// TIA Portal project "Parcel-locker-siemensS7" (V16)

(* hardware
DEVICE "S71500/ET200MP station_1"  S7-1500 station
   slot 0: "Rail_0"  Rack  6ES7 590-1***0-0AA0
   slot 1: "PLC_1"  CPU 1512C-1 PN  6ES7 512-1CK01-0AB0  V2.8
      slot 3: "CPU display_1"  6ES7591-1AA00-0AA0
      slot 32768: "PROFINET interface_1"  X1
         slot 32769: "Port_1"  X1 P1
         slot 32770: "Port_2"  X1 P2
      slot 34817: "Virtual CP interface port_1"  Virtual CP interface port  Virtual CP interface port
*)

// ===== PLC "PLC_1"  CPU 1512C-1 PN =====

VAR_GLOBAL   // PLC tag table "Default tag table"
   "Box1" AT %Q0.0 : Bool;
   "Box2" AT %Q0.1 : Bool;
   "Box3" AT %Q0.2 : Bool;
END_VAR

// folder: Common

TYPE "typeDiagnostics"
TITLE = typeDiagnostics
// Provides a structure for detailed diagnostics
   STRUCT
      status : Word;   // Status of the block or error identification when error occurred
      subfunctionStatus : DWord;   // Status or return value of called FBs, FCs and system blocks
      stateNumber : DInt;   // State in the state machine of the block where the error occurred
   END_STRUCT;
END_TYPE

// folder: LHTTP

TYPE "LHTTP_typeTLS"
   STRUCT
      validateServerIdentity : Bool;   // Validate the subjectAlternateName in the X.509-V3 certificate of the server to check the identity of the server
      serverCert : UDInt;   // ID of the X.509-V3 certificate (usually a CA certificate) that is used by the TLS client to validate the TLS server authentication. If this parameter is 0, the TLS client uses all (CA) certificates currently loaded in the client certificate store to validate the server authentication.
      clientCert : UDInt;   // ID of own X.509 V3 certificate
   END_STRUCT;
END_TYPE

// folder: (top level)

DATA_BLOCK "Modbus_server_parameters"   // DB2
{ S7_Optimized_Access := 'TRUE' }
VERSION : 0.1
   VAR
      NDR : Bool;
      DR : Bool;
      ERROR : Bool;
      STATUS : Word;
      CONNECT : TCON_IP_v4;
   END_VAR
BEGIN
   CONNECT.InterfaceId := 64;
   CONNECT.ID := 1;
   CONNECT.LocalPort := 502;
END_DATA_BLOCK

DATA_BLOCK "Modbus_data"   // DB3
{ S7_Optimized_Access := 'FALSE' }
VERSION : 0.1
   VAR
      Boxes : Array[0..3] of Int;
   END_VAR
BEGIN
END_DATA_BLOCK

DATA_BLOCK "Modbus_server_DB"   // DB4
{ S7_Optimized_Access := 'TRUE' }
VERSION : 0.1
// stored: InstanceOfName Modbus_server
"Modbus_server"
BEGIN
END_DATA_BLOCK

FUNCTION_BLOCK "Modbus_server"   // FB1, LAD
{ S7_Optimized_Access := 'TRUE' }
VERSION : 0.1
BEGIN

REGION Network 1
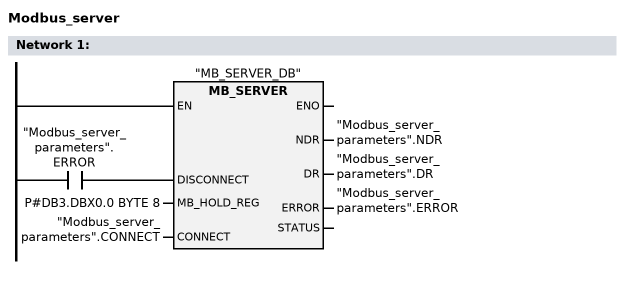
   "MB_SERVER_DB"(DISCONNECT := "Modbus_server_parameters".ERROR,   // MB_SERVER
                  MB_HOLD_REG := P#DB3.DBX0.0 BYTE 8,
                  CONNECT := "Modbus_server_parameters".CONNECT,
                  NDR => "Modbus_server_parameters".NDR,
                  DR => "Modbus_server_parameters".DR,
                  ERROR => "Modbus_server_parameters".ERROR);
END_REGION
END_FUNCTION_BLOCK

ORGANIZATION_BLOCK "Main"   // OB1, LAD, ProgramCycle
TITLE = "Main Program Sweep (Cycle)"
{ S7_Optimized_Access := 'TRUE' }
VERSION : 0.1
   VAR_INPUT
      Initial_Call : Bool;   // Initial call of this OB
      Remanence : Bool;   // =True, if remanent data are available
   END_VAR
BEGIN

REGION Network 1
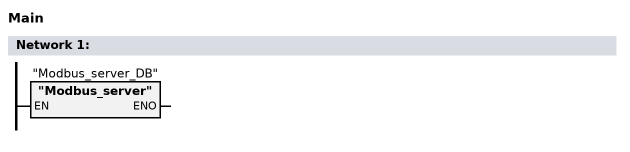
   RUNG wire#powerrail
      "Modbus_server_DB"()
   END_RUNG
   // the same network as SCL:
   "Modbus_server_DB"();   // "Modbus_server"
END_REGION

REGION Network 3 (SCL)
   // Open Box1
   IF ("Modbus_data".Boxes[0] AND 2#0000_0000_0000_0001) <> 0 THEN
       "Box1" := TRUE;
   ELSE
       "Box1" := FALSE;
   END_IF;
END_REGION

REGION Network 4 (SCL)
   // Open Box2
   IF ("Modbus_data".Boxes[0] AND 2#0000_0000_0000_0010) <> 0 THEN
       "Box2" := TRUE;
   ELSE
       "Box2" := FALSE;
   END_IF;
END_REGION

REGION Network 5 (SCL)
   // Open Box3
   IF ("Modbus_data".Boxes[0] AND 2#0000_0000_0000_0100) <> 0 THEN
       "Box3" := TRUE;
   ELSE
       "Box3" := FALSE;
   END_IF;
END_REGION
END_ORGANIZATION_BLOCK

// ===== library types =====

// folder: LHTTP

FUNCTION_BLOCK "LHTTP_Get"   // FB8, SCL
TITLE = LHTTP_Get
{ S7_Optimized_Access := 'TRUE' }
AUTHOR : SIOS
FAMILY : LHTTP
VERSION : 2.1
// Implements the HTTP GET method
   VAR_INPUT
      execute : Bool;   // Send HTTP request
      hwID : Hw_Any;   // Hardware ID of Ethernet interface
      connID : Conn_Ouc := 1;   // Unique connection ID
      url : String;   // URL, i.e. "http://www.siemens.com/simatic"
      queryParams : String;   // Additional query parameters if "url" is not long enough, i.e. "lang=en&q=simatic"; "?" or "&" is inserted automatically in between "url" and "queryParameters". / Optional query parameters that are appended to URL, i.e. "lang=en&q=simatic"
      userFields : Array[0..#UPPER_USER_FIELDS] of Char;   // Additional user-defined header fields
      tls : "LHTTP_typeTLS";   // TLS certificates for secure connections (HTTPS), leave open for non-secure connections (HTTP)
      keepConnection : Bool;   // Keep connection established after execution of request
      timeOut : Time := T#10s;   // Time to wait for response from server
   END_VAR
   VAR_OUTPUT
      connected : Bool;   // Connection to web server is established
      done : Bool;   // HTTP request finished
      busy : Bool;   // Function is busy
      error : Bool;   // An error occured
      status : Word := 16#7000;   // Specifies the error
      diagnostics : "typeDiagnostics";   // Diagnostics information of FB
      responseCode : UInt;   // HTTP response code
      length : UDInt;   // Length of received data
   END_VAR
   VAR_IN_OUT
      responseData : Array[*] of Char;   // Data received from HTTP server
   END_VAR
   VAR
      instTSendC : TSEND_C;   // Instance of TSEND_C
      instTRcv : TRCV;   // Instance of TRCV
      instTimeout : TON_TIME;   // Time-out
      statConnected : Bool;   // Static value for output 'connected'
      statDone : Bool;   // Static value for output 'done'
      statBusy : Bool;   // Static value for output 'busy'
      statError : Bool;   // Static value for output 'error'
      statStatus : Word := 16#7000;   // Static value for output 'status'
      statResponseCode : UInt;   // Static value for output 'responseCode'
      statLength : UDInt;   // Static value for output 'length'
      statFBState : USInt := 0;   // Current state in state machine
      statSubfunctionStatus : DWord;   // Status or return value of called FBs, FCs and system blocks
      statEmptyDiagnostics : "typeDiagnostics";   // Empty diagnostics information (for initialization purposes only)
      statParam : Struct   // Connection parameters
         isQDN : Bool;
         paramQDN : TCON_QDN_SEC;   // Connection parameters in form of QDN
         paramIP : TCON_IP_V4_SEC;   // Connection parameters in form of IP address
      END_STRUCT;
      statHost : String;   // Host part of URL
      statRequest : Struct   // GET request
         chars : Array[0..#UPPER_REQUEST_ARRAY] of Char;   // GET request (max. length: url (254) + data (254) + header (94)
         length : UInt;   // Length of GET request
      END_STRUCT;
      statSend : Struct   // Parameters for instruction TSend_C
         connect : Bool;   // Establish and keep connection
         req : Bool;   // Send data
      END_STRUCT;
      statEncoding : String;   // Transfer encoding of response from HTTP server
      statContentLength : UInt;   // Content length as specified in header of response
      statChunkLen : UDInt;   // Remaining length of current chunk
      statRcvdLen : UDInt;   // Sum length of received data
      statTimeoutIn : Bool;   // Timeout
      statRcvBuffer : Array[0..#UPPER_TCP_FRAME] of Char;   // Temporary receive buffer
      statSizeRcvArray : UDInt;   // Size of receive buffer at parameter "responseData"
      statExecuteOld : Bool;   // Last cycle's value of input "execute"
   END_VAR
   VAR_TEMP
      tempUrl : String;   // Copy of URL
      tempQuery : String;   // Query part of URL
      tempIndex : DInt;   // Index for for loops
      tempPos : Int;   // General tag for positions
      tempLen : UInt;   // General tag for lengths
      tempRet : Word;   // General tag for return values
      tempString : String;   // General tag for strings
      tempExitLoop : Bool;   // Condition to exit REPEAT loop around state machine
      tempChunk : Struct   // Temporary tags for chunked encoding
         posData : UInt;   // Start position of data in current packet
         lenData : UInt;   // Length of data in current packet
         exitLoop : Bool;   // Condition to exit loop
      END_STRUCT;
   END_VAR
   VAR CONSTANT
      UPPER_REQUEST_ARRAY : UInt := 1459;   // Upper limit of request array
      UPPER_TCP_FRAME : UInt := 1459;   // Upper limit of a TCP/IP frame
      UPPER_USER_FIELDS : USInt := 255;   // Upper limit of userFields
      PORT_UNSECURE : UInt := 80;   // Port for unsecure HTTP connection
      PORT_SECURE : UInt := 443;   // Port for secure HTTP connection
      POS_RESPONSE_CODE : USInt := 9;   // Position of HTTP response code in response message
      STATUS_DONE : Word := 16#0000;   // Job finished without errors
      STATUS_DISCONNECTED : Word := 16#0003;   // Communication connection closed
      STATUS_IDLE : Word := 16#7000;   // No job
      STATUS_FIRST_CALL : Word := 16#7001;   // First call after incoming new job (rising edge 'execute')
      STATUS_CONNECTING : Word := 16#7002;   // Connection is currently being established
      STATUS_DISCONNECTING : Word := 16#7003;   // Communication connection is being terminated
      STATUS_MONITORING : Word := 16#7004;   // Communication connection has been established and is being monitored. No send job execution active
      STATUS_SENT : Word := 16#7005;   // Request sent, waiting for response
      SUB_STATUS_NO_ERROR : DWord := 16#0000_0000;   // No error occured in subfunction call
      ERR_BOUND_NOT_ZERO : Word := 16#8201;   // Lower bound of receive buffer is not 0
      ERR_INVALID_URL : Word := 16#8202;   // Invalid URL
      ERR_DIFFERENT_HOST : Word := 16#8203;   // Trying to use existing connection with different host
      ERR_END_USER_FIELDS : Word := 16#8206;   // End of user-defined header fields could not be found
      ERR_REQUEST_SIZE : Word := 16#8210;   // Request array is too small for specified parameters
      ERR_RESPONSE_SIZE : Word := 16#8220;   // Receive buffer at parameter "responseData" too small
      ERR_CONN_LOST : Word := 16#8400;   // Offset for lost connection
      ERR_FORWARDING : Word := 16#8403;   // Server responded with forwarding message. Forwarding is not supported, see "diagnostics"
      ERR_WEBSERVER : Word := 16#8404;   // Webserver responded with error code, see "diagnostics"
      ERR_INVALID_HEADER : Word := 16#8405;   // Header of response is invalid
      ERR_TIMEOUT : Word := 16#8408;   // Time-out occurred
      ERR_UNDEFINED_STATE : Word := 16#8600;   // Error due to an undefined state in state machine
      ERR_TSENDC : Word := 16#8601;   // Error: TCON encountered an error, see "diagnostics"
      ERR_TRCV : Word := 16#8603;   // Error: TURCV encountered error, see "diagnostics"
      ERR_MOVE_USER_FIELDS : Word := 16#8612;   // Error in MOVE_BLK_VARIANT to copy user-defined header fields, see "diagnostics"
      ERR_ENCODING_UNKNOWN : Word := 16#8620;   // Transfer encoding of response could not be detected or is unsupported
      ERR_MOVE_IDENTITY : Word := 16#8630;   // Error in MOVE_BLK_VARIANT for transfer encoding 'identity', see "diagnostics"
      ERR_DECODING_FAILED : Word := 16#8640;   // Chunk encoded response could not be decoded
      ERR_MOVE_CHUNKED : Word := 16#8641;   // Error in MOVE_BLK_VARIANT for transfer encoding 'chunked', see "diagnostics"
      TSENDC_STATUS_CONNECTED : Word := 16#0001;   // TSEND_C: Communication connection established
      MOVE_STATUS_SIZE : Word := 16#8483;   // MOVE_BLK_VARIANT: DEST too small
      FB_STATE_NO_PROCESSING : USInt := 0;   // FB state: No processing
      FB_STATE_INIT : USInt := 1;   // FB state: initialization
      FB_STATE_REQUEST : USInt := 2;   // FB state: prepare request
      FB_STATE_SEND : USInt := 3;   // FB state: send request
      FB_STATE_RCV : USInt := 4;   // FB state: receive data
      FB_STATE_MON : USInt := 5;   // FB state: monitoring connection
      CRLF : String := '$R$L';   // Newline control character (carriage return, line feed)
      HEADER_END : String := '$R$L$R$L';   // End of HTTP header (two newline control characters)
      LEN_CRLF : UInt := 2;   // Length of CRLF
   END_VAR
   // statParam.paramIP.ConnPara.ActiveEstablished := true;
   // statParam.paramQDN.ConnPara.ActiveEstablished := true;
BEGIN
   REGION BLOCK INFO HEADER
     //===============================================================================
     // SIEMENS / (c)Copyright 2021
     //-------------------------------------------------------------------------------
     // Title:        LHTTP_Get
     // Function:     Implements the HTTP GET method
     // Library:      LHTTP
     // Author:       Siemens Industry Online Support
     // Tested with:  CPU 1516-3 PN/DP V2.8
     // Engineering:  TIA Portal V16
     // Restrictions: --
     // Requirements: S7-1200 with firmware V4.4 or higher
     //               S7-1500 with firmware V2.0 or higher
     //-------------------------------------------------------------------------------
     // Change log table:
     // Version  | Date       | Expert in charge       | Changes applied
     //----------|------------|------------------------|------------------------------
     // 02.01.00 | 2021-12-15 | Online Support         | Renamed parameter "data" to "queryParams"
     //-------------------------------------------------------------------------------
     // 02.00.04 | 2021-05-10 | Online Support         | Fixed issues with chunked encoding
     //          |            |                        | Allow chunk sizes > 65535 Bytes
     //          |            |                        | Made header evaluation case-insensitive
     //-------------------------------------------------------------------------------
     // 02.00.00 | 2020-12-16 | Online Support         | Added option to keep connection established
     //          |            |                        | Added parameter to add user-defined headers fields
     //          |            |                        | Changed to data type of "data" to Variant to allow larger data
     //          |            |                        | Removed "statusID" and added "diagnostics" instead, changed some error codes
     //-------------------------------------------------------------------------------
     // 01.00.00 | 2019-04-01 | Online Support         | First released version
     //===============================================================================
   END_REGION

   REGION INSTRUCTIONS
     IF (#statStatus <> #STATUS_IDLE) THEN // Only execute when FB is triggered to reduce system load
       // Connect and send
       IF #statParam.isQDN THEN // Call if host is a domain name
         #instTSendC(REQ     := #statSend.req,
                     CONT    := #statSend.connect,
                     LEN     := #statRequest.length,
                     CONNECT := #statParam.paramQDN,
                     DATA    := #statRequest.chars);
       ELSE // Call if host is an IP address
         #instTSendC(REQ     := #statSend.req,
                     CONT    := #statSend.connect,
                     LEN     := #statRequest.length,
                     CONNECT := #statParam.paramIP,
                     DATA    := #statRequest.chars);
       END_IF;

       // Receive
       #instTRcv(ID    := #statParam.paramQDN.ConnPara.ID,
                 EN_R  := #statFBState >= #FB_STATE_RCV,
                 LEN   := 0,
                 ADHOC := true,
                 DATA  := #statRcvBuffer);

       // Monitor time out
       #instTimeout(IN := #statTimeoutIn,
                    PT := #timeOut);

       IF #instTimeout.Q THEN
         #statStatus := #ERR_TIMEOUT;
       END_IF;
     END_IF;
   END_REGION

   REGION TRIGGERING
     IF (#execute = true AND #statExecuteOld = false) // Check if FB is triggered
       AND (#statStatus = #STATUS_IDLE OR #statStatus = #STATUS_MONITORING)
     THEN // First call; initialize FB
       // Copy URL
       #tempUrl := #url;

       #statBusy := true;
       #statStatus := #STATUS_FIRST_CALL;
       #statSubfunctionStatus := #SUB_STATUS_NO_ERROR;
       #diagnostics := #statEmptyDiagnostics;

       IF #statConnected = FALSE THEN // Connection is not yet established
         #statFBState := #FB_STATE_INIT;
       ELSE // Connection is already established, skip init
         #statFBState := #FB_STATE_REQUEST;
       END_IF;

     ELSIF (#statStatus = #STATUS_FIRST_CALL) THEN
       #statStatus := #STATUS_CONNECTING;
     END_IF;

     // Edge detection 'execute' input
     #statExecuteOld := #execute;
   END_REGION TRIGGERING

   IF (#statStatus = #STATUS_IDLE) THEN // Nothing to do -> End here to reduce "system load"
     RETURN;
   END_IF;

   REGION STATE_MACHINE
     // State machine is wrapped in REPEAT loop to make it possible to quickly exit state machine
     // in case of an error or to go through CASE multiple times within one cycle
     REPEAT
       #tempExitLoop := true; // Condition to exit loop is set per default

       CASE #statFBState OF // State machine of FB
         #FB_STATE_NO_PROCESSING: // No processing active
           ;

         #FB_STATE_INIT:
           REGION INIT
             // Get size of receive buffer
             IF LOWER_BOUND(ARR := #responseData, DIM := 1) <> 0 THEN
               #statStatus := #ERR_BOUND_NOT_ZERO;
               EXIT;
             ELSE
               #statSizeRcvArray := DINT_TO_UDINT(UPPER_BOUND(ARR := #responseData, DIM := 1)) + 1;
             END_IF;

             // Set connection parameters
             #statParam.paramQDN.ConnPara.InterfaceId := #hwID;
             #statParam.paramQDN.ConnPara.ID := #connID;
             #statParam.paramIP.ConnPara.InterfaceId := #hwID;
             #statParam.paramIP.ConnPara.ID := #connID;

             // Check if network protocol was specified to determine if connection should be secured
             #tempPos := FIND(IN1 := #tempUrl, IN2 := 'https://');
             IF #tempPos = 1 THEN // HTTPS
               #statParam.paramQDN.ActivateSecureConn := true;
               #statParam.paramQDN.ExtTLSCapabilities.%X0 := #tls.validateServerIdentity;
               #statParam.paramQDN.TLSServerCertRef := #tls.serverCert;
               #statParam.paramQDN.TLSClientCertRef := #tls.clientCert;
               #statParam.paramIP.ActivateSecureConn := true;
               #statParam.paramIP.ExtTLSCapabilities.%X0 := #tls.validateServerIdentity;
               #statParam.paramIP.TLSServerCertRef := #tls.serverCert;
               #statParam.paramIP.TLSClientCertRef := #tls.clientCert;
               // Delete network protocol from URL
               #tempUrl := DELETE(IN := #tempUrl, L := 8, P := 1);
             ELSE // HTTP
               #statParam.paramQDN.ActivateSecureConn := false;
               #statParam.paramIP.ActivateSecureConn := false;
               // Delete network protocol from URL if specified
               IF #tempUrl[5] = ':' THEN
                 #tempUrl := DELETE(IN := #tempUrl, L := 7, P := 1);
               END_IF;
             END_IF;

             // Determine if host is domain name or IP address
             #tempPos := CHAR_TO_INT(#tempUrl[1]);
             IF #tempPos >= CHAR_TO_INT('A') AND #tempPos <= CHAR_TO_INT('z') THEN // Host is a domain name
               #statParam.isQDN := true;
             ELSIF #tempPos >= CHAR_TO_INT('0') AND #tempPos <= CHAR_TO_INT('9') THEN // Host is an IP address
               #statParam.isQDN := false;
             ELSE // URL invalid
               #statStatus := #ERR_INVALID_URL;
               EXIT;
             END_IF;

             // Get host name and port
             #tempPos := FIND(IN1 := #tempUrl, IN2 := '/');
             IF #tempPos > 0 THEN // URL has a path after host name
               #statHost := LEFT(IN := #tempUrl, L := #tempPos - 1);
             ELSE
               #statHost := #tempUrl;
             END_IF;
             #tempPos := FIND(IN1 := #statHost, IN2 := ':');
             IF #tempPos > 0 THEN // Port specified in URL
               #statParam.paramQDN.ConnPara.RemotePort := STRING_TO_UINT(DELETE(IN := #statHost, L := #tempPos, P := 1));
               #statParam.paramIP.ConnPara.RemotePort := STRING_TO_UINT(DELETE(IN := #statHost, L := #tempPos, P := 1));
               #statHost := LEFT(IN := #statHost, L := #tempPos - 1);
             ELSE // No port specified in URL, set default port
               IF #statParam.paramQDN.ActivateSecureConn OR #statParam.paramIP.ActivateSecureConn THEN
                 #statParam.paramQDN.ConnPara.RemotePort := #PORT_SECURE;
                 #statParam.paramIP.ConnPara.RemotePort := #PORT_SECURE;
               ELSE
                 #statParam.paramQDN.ConnPara.RemotePort := #PORT_UNSECURE;
                 #statParam.paramIP.ConnPara.RemotePort := #PORT_UNSECURE;
               END_IF;
             END_IF;

             IF #statParam.isQDN THEN // Host is a domain name
               #statParam.paramQDN.ConnPara.RemoteQDN := CONCAT(IN1 := #statHost, IN2 := '.');
             ELSE // Host is an IP address
               #tempString := #statHost;
               FOR #tempIndex := 1 TO 3 DO
                 #tempPos := FIND(IN1 := #tempString, IN2 := '.');
                 #statParam.paramIP.ConnPara.RemoteAddress.ADDR[#tempIndex] := UINT_TO_BYTE(STRING_TO_UINT(LEFT(IN := #tempString, L := #tempPos - 1)));
                 #tempString := DELETE(IN := #tempString, L := #tempPos, P := 1);
               END_FOR;
               #statParam.paramIP.ConnPara.RemoteAddress.ADDR[4] := UINT_TO_BYTE(STRING_TO_UINT(#tempString));
             END_IF;

             #statFBState := #FB_STATE_REQUEST;
             #tempExitLoop := FALSE; // Don't exit loop to go directly to prepare request
           END_REGION INIT

         #FB_STATE_REQUEST:
           REGION PREP_REQUEST
             // Check host in URL when using existing connection
             IF #statConnected = TRUE THEN
               #tempPos := FIND(IN1 := #tempUrl, IN2 := #statHost);
               IF #tempPos = 0 THEN // URL doesn't contain expected host
                 #statStatus := #ERR_DIFFERENT_HOST;
                 EXIT;
               ELSE // Scheme and host must be deleted for further processing
                 #tempUrl := DELETE(IN := #tempUrl, L := #tempPos + LEN(#statHost) - 1, P := 1);
               END_IF;
             END_IF;

             // Get path
             #tempPos := FIND(IN1 := #tempUrl, IN2 := '/');
             IF #tempPos > 0 THEN // URL has a path after host name
               #tempString := DELETE(IN := #tempUrl, L := #tempPos - 1, P := 1);
             ELSE
               #tempString := '/';
             END_IF;

             // Prepare query part of URL
             IF #queryParams <> '' THEN // Parameter is in use
               IF #queryParams[1] = '?' OR #queryParams[1] = '&' THEN
                 #tempQuery := DELETE(IN := #queryParams, P := 1, L := 1);
               ELSE
                 #tempQuery := #queryParams;
               END_IF;
               #tempPos := FIND(IN1 := #tempString, IN2 := '?'); // Check if URL already contains query parameters
               IF #tempPos <> 0 THEN // URL already contains query parameters
                 #tempQuery := CONCAT(IN1 := '&', IN2 := #tempQuery); // Append query parameters with &
               ELSE // URL does not contain query parameters
                 #tempQuery := CONCAT(IN1 := '?', IN2 := #tempQuery); // Append query parameters with ?
               END_IF;
             END_IF;

             // Put together GET request
             // Strg_TO_Chars conversion is done several times to utilize maximum length of parameters url and query parameters
             Strg_TO_Chars(Strg   := CONCAT(IN1 := 'GET ', IN2 := #tempString), // Path cannot be longer than 249 characters --> save to use CONCAT
                           pChars := 0,
                           Cnt    => #tempLen,
                           Chars  := #statRequest.chars);
             #tempPos := UINT_TO_INT(#tempLen);

             Strg_TO_Chars(Strg   := #tempQuery,
                           pChars := #tempPos,
                           Cnt    => #tempLen,
                           Chars  := #statRequest.chars);
             #tempPos += UINT_TO_INT(#tempLen);

             Strg_TO_Chars(Strg   := CONCAT(IN1 := ' HTTP/1.1$R$LHost: ', IN2 := #statHost), // Host will not use all 254 characters --> save to use CONCAT
                           pChars := #tempPos,
                           Cnt    => #tempLen,
                           Chars  := #statRequest.chars);
             #tempPos += UINT_TO_INT(#tempLen);

             Strg_TO_Chars(Strg   := '$R$LUser-Agent: SIMATIC Controller (LHTTP)$R$LAccept: text/html$R$LAccept-Encoding: identity$R$LAccept-Charset: utf-8$R$L',
                           pChars := #tempPos,
                           Cnt    => #tempLen,
                           Chars  := #statRequest.chars);
             #tempPos += UINT_TO_INT(#tempLen);

             // Insert additional user-defined header fields
             IF #userFields[0] <> ' ' THEN
               FOR #tempLen := 0 TO #UPPER_USER_FIELDS DO
                 IF #userFields[#tempLen] = '$00' THEN
                   EXIT;
                 END_IF;
               END_FOR;

               IF #tempLen > #UPPER_USER_FIELDS THEN // End not found
                 #statStatus := #ERR_END_USER_FIELDS;
                 EXIT;
               END_IF;

               #tempRet := INT_TO_WORD(MOVE_BLK_VARIANT(SRC := #userFields, COUNT := #tempLen, SRC_INDEX := 0, DEST_INDEX := #tempPos, DEST => #statRequest.chars));

               IF #tempRet = #MOVE_STATUS_SIZE THEN
                 #statStatus := #ERR_REQUEST_SIZE;
                 EXIT;
               ELSIF #tempRet <> 16#0000 THEN
                 #statStatus := #ERR_MOVE_USER_FIELDS;
                 #statSubfunctionStatus := #tempRet;
                 EXIT;
               END_IF;

               #tempPos += UINT_TO_INT(#tempLen);

               // Append CRLF if needed
               IF #statRequest.chars[#tempPos - 2] <> '$R' AND #statRequest.chars[#tempPos - 1] <> '$L' THEN
                 #statRequest.chars[#tempPos] := '$R';
                 #statRequest.chars[#tempPos + 1] := '$L';
                 #tempPos += 2;
               END_IF;
             END_IF;

             // Append end of header section
             Strg_TO_Chars(Strg   := #CRLF,
                           pChars := #tempPos,
                           Cnt    => #tempLen,
                           Chars  := #statRequest.chars);
             #tempPos += UINT_TO_INT(#tempLen);

             // Calculate total length of request
             #statRequest.length := INT_TO_UINT(#tempPos);

             #statSend.connect := true; // Connect
             #statSend.req := true; // Send request
             #statTimeoutIn := true; // Start timer
             #statFBState := #FB_STATE_SEND;
           END_REGION

         #FB_STATE_SEND: // Send data
           REGION SEND
             IF #instTSendC.STATUS = #TSENDC_STATUS_CONNECTED THEN
               #statConnected := TRUE;
             ELSIF #instTSendC.DONE THEN
               #statStatus := #STATUS_SENT;
               #statFBState := #FB_STATE_RCV;
               // Don't exit loop to go directly to receive state
               // without waiting for next cycle so that no responses can be missed
               #tempExitLoop := false;
             ELSIF #instTSendC.ERROR THEN
               #statStatus := #ERR_TSENDC;
               #statSubfunctionStatus := #instTSendC.STATUS;
             END_IF;
           END_REGION

         #FB_STATE_RCV: // Wait for new data
           REGION RCV
             IF #instTRcv.NDR THEN

               REGION HEADER_EVAL
                 // Evaluate header if received packet is first packet
                 IF #statEncoding = '' THEN
                   // Get response code
                   Chars_TO_Strg(Chars  := #statRcvBuffer,
                                 pChars := #POS_RESPONSE_CODE,
                                 Cnt    := 3,
                                 Strg   => #tempString);
                   #statResponseCode := STRING_TO_UINT(#tempString);

                   // Exit loop immediately and output errror if response code shows errors or forwarding
                   IF #statResponseCode >= 300 THEN
                     #tempRet := ATH(IN := #tempString, N := 3, OUT => #statSubfunctionStatus); // Interpret response code as hexadecimal
                     #statSubfunctionStatus := SHR(IN := #statSubfunctionStatus, N := 20);
                     IF #statResponseCode >= 400 THEN
                       #statStatus := #ERR_WEBSERVER;
                     ELSE
                       #statStatus := #ERR_FORWARDING;
                     END_IF;
                     EXIT;
                   END_IF;

                   // Get length of HTTP header
                   #tempLen := DINT_TO_UINT("LHTTP_FindStringInArray"(searchFor := #HEADER_END, searchIn := #statRcvBuffer) + LEN(#HEADER_END));

                   // Exit loop immediately and output errror if header end cannot be found
                   IF #tempLen = 0 THEN
                     #statStatus := #ERR_INVALID_HEADER;
                     EXIT;
                   END_IF;

                   // Search header for content length
                   #tempRet := "LHTTP_ExtractStringFromArray"(textBefore := 'Content-Length: ',
                                                              textAfter := #CRLF,
                                                              extractedString => #tempString,
                                                              searchIn := #statRcvBuffer);

                   IF #tempRet <> 0 THEN // Content length not found; try lower-case
                     #tempRet := "LHTTP_ExtractStringFromArray"(textBefore := 'content-length: ',
                                                                textAfter := #CRLF,
                                                                extractedString => #tempString,
                                                                searchIn := #statRcvBuffer);
                   END_IF;

                   IF #tempRet = 0 THEN // Content length found
                     #statContentLength := STRING_TO_UINT(#tempString);
                     #statEncoding := 'identity';
                   ELSE // Can't detect content length, check if transfer encoding is 'chunked'
                     #tempPos := DINT_TO_INT("LHTTP_FindStringInArray"(searchFor := 'chunked', searchIn := #statRcvBuffer));

                     IF #tempPos >= 0 THEN
                       #statEncoding := 'chunked';
                     ELSE // Exit loop immediately and output error if content length nor transfer encoding can be detected
                       #statStatus := #ERR_ENCODING_UNKNOWN;
                       EXIT;
                     END_IF;
                   END_IF;

                   IF #instTRcv.RCVD_LEN = #tempLen THEN // Packet contains no body, wait for next packet
                     EXIT;
                   END_IF;
                 END_IF;
               END_REGION

               REGION TE_IDENTITY
                 IF #statEncoding = 'identity' THEN // Transfer encoding is 'identity'
                   // Move data from buffer to output; tempLen contains header length during first packet, otherwise 0
                   #tempRet := INT_TO_WORD(MOVE_BLK_VARIANT(SRC := #statRcvBuffer,
                                                                                    COUNT := MIN(IN1 := #instTRcv.RCVD_LEN - #tempLen, IN2 := #statSizeRcvArray - #statRcvdLen), // Move as much as possible to output
                                                                                    SRC_INDEX := #tempLen,
                                                                                    DEST_INDEX := UDINT_TO_DINT(#statRcvdLen),
                                                                                    DEST => #responseData));

                   // Exit loop immediately and output error if data could not be moved
                   IF #tempRet <> 0 THEN
                     #statStatus := #ERR_MOVE_IDENTITY;
                     #statSubfunctionStatus := #tempRet;
                     EXIT;
                   END_IF;

                   // Add length of received packet to sum; tempLen contains header length during first packet, otherwise 0
                   #statRcvdLen += #instTRcv.RCVD_LEN - #tempLen;

                   IF #statRcvdLen > #statSizeRcvArray THEN // Receive buffer too small
                     #statStatus := #ERR_RESPONSE_SIZE;
                     #statLength := #statContentLength; // Output required size of buffer
                   ELSIF #statRcvdLen >= #statContentLength THEN // Everything was received
                     #statStatus := #STATUS_DONE;
                     #statLength := #statRcvdLen;
                   END_IF;
                 END_IF;
               END_REGION

               REGION TE_CHUNKED
                 IF #statEncoding = 'chunked' THEN // Transfer encoding is 'chunked'

                   // Set position of chunk data
                   #tempChunk.posData := #tempLen; // tempLen contains header length during first packet, otherwise 0

                   REPEAT
                     #tempChunk.exitLoop := true; // Condition to exit loop is set per default

                     // Read length of chunk if received packet is first packet or a previous chunk was received completely
                     IF #statChunkLen = 0 THEN
                       // Extract hexadecimal chunk-size field
                       Chars_TO_Strg(Chars  := #statRcvBuffer,
                                     pChars := #tempChunk.posData,
                                     Cnt    := 0,
                                     Strg   => #tempString);
                       #tempPos := FIND(IN1 := #tempString, IN2 := #CRLF);
                       #tempRet := ATH(IN := #tempString, N := #tempPos - 1, OUT => #statChunkLen);
                       // Shift bits to the right depending on length of chunk size, since ATH is left aligned
                       #statChunkLen := SHR(IN := #statChunkLen, N := 4 * INT_TO_UINT(8 - (#tempPos - 1)));

                       // Move start position of data behind chunk-size field
                       #tempChunk.posData += INT_TO_UINT(#tempPos) + 1;

                       // Exit loop immediately and output error if chunk size cannot be detected
                       IF #tempRet <> 0 THEN
                         #statStatus := #ERR_DECODING_FAILED;
                         EXIT;
                       END_IF;
                     END_IF;

                     IF #statChunkLen = 0 THEN // Length was evaluated, chunk contains no data --> final chunk received
                       #statStatus := #STATUS_DONE;
                       #statLength := #statRcvdLen;
                     ELSE // Chunk contains data
                       // Evaluate length of received packet and set length of data accordingly
                       IF #instTRcv.RCVD_LEN = #tempChunk.posData + #statChunkLen + #LEN_CRLF THEN // Chunk was received entirely and packet contains no further chunks
                         #tempChunk.lenData := UDINT_TO_UINT(#statChunkLen); // Output remaining length of chunk
                       ELSIF #instTRcv.RCVD_LEN < #tempChunk.posData + #statChunkLen + #LEN_CRLF THEN // Packet only contains part of chunk
                         #tempChunk.lenData := UDINT_TO_UINT(#instTRcv.RCVD_LEN) - #tempChunk.posData; // Output entire packet without possible chunk-size field
                       ELSIF #instTRcv.RCVD_LEN > #tempChunk.posData + #statChunkLen + #LEN_CRLF THEN // Current packet contains more than one chunk
                         #tempChunk.lenData := UDINT_TO_UINT(#statChunkLen); // Output remaining length of chunk
                         #tempChunk.exitLoop := false; // Execute loop again since packet contains more data
                       ELSE // Can't decode message
                         #statStatus := #ERR_DECODING_FAILED;
                         EXIT;
                       END_IF;

                       // Move received data to output
                       #tempRet := INT_TO_WORD(MOVE_BLK_VARIANT(SRC := #statRcvBuffer,
                                                                                        COUNT := MIN(IN1 := #tempChunk.lenData, IN2 := #statSizeRcvArray - #statRcvdLen), // Move as much as possible to output
                                                                                        SRC_INDEX := #tempChunk.posData,
                                                                                        DEST_INDEX := UDINT_TO_DINT(#statRcvdLen),
                                                                                        DEST => #responseData));

                       // Exit loop immediately and output error if data could not be moved
                       IF #tempRet <> 0 THEN
                         #statStatus := #ERR_MOVE_CHUNKED;
                         #statSubfunctionStatus := #tempRet;
                         EXIT;
                       END_IF;

                       // Move start position of data behind data of current chunk in case packet contains more data; only relevant if REPEAT loop is executed again
                       #tempChunk.posData += #tempChunk.lenData + #LEN_CRLF;

                       // Subtract length of data in current packet from remaining length of chunk and add to sum of received data
                       #statChunkLen -= #tempChunk.lenData;
                       #statRcvdLen += #tempChunk.lenData;

                       IF #statRcvdLen > #statSizeRcvArray THEN // Receive buffer too small
                         #statStatus := #ERR_RESPONSE_SIZE;
                         #statLength := #statRcvdLen; // Output required size of buffer according to so far received chunked messages
                         EXIT;
                       END_IF;
                     END_IF;
                   UNTIL (#tempChunk.exitLoop = true) END_REPEAT;
                 END_IF;
               END_REGION

             ELSIF #instTRcv.ERROR THEN
               #statStatus := #ERR_TRCV;
               #statSubfunctionStatus := #instTRcv.STATUS;
             END_IF;
           END_REGION

         #FB_STATE_MON:
           REGION MONITORING
             IF #keepConnection = FALSE THEN // Trigger to disconnect
               #statSend.connect := FALSE;
               #statDone := FALSE;
               #statBusy := TRUE;
               #statStatus := #STATUS_DISCONNECTING;
             END_IF;

             IF #instTSendC.STATUS = #STATUS_DISCONNECTED THEN
               #statConnected := FALSE;
               #statStatus := #STATUS_DISCONNECTED;
             ELSIF #instTRcv.ERROR THEN
               #statConnected := FALSE;
               #statStatus := #ERR_CONN_LOST OR (#instTRcv.STATUS AND 16#00FF);
             END_IF;
           END_REGION

         ELSE // Undefined state in state machine reached
           #statStatus := #ERR_UNDEFINED_STATE;
       END_CASE;

     UNTIL (#tempExitLoop = true) END_REPEAT;
   END_REGION

   REGION OUTPUTS
     // Write outputs
     IF (#statStatus = #STATUS_DONE) AND (#statDone = false) THEN // Execution finished without errors
       #statDone := true;
       #statBusy := false;
       #statError := false;
       #statSend.connect := #keepConnection;
       #statSend.req := false;
       #statTimeoutIn := false;

       IF #keepConnection THEN
         // execution finished but connection is kept alive --> set state monitoring
         #statFBState := #FB_STATE_MON;
       ELSE
         #statConnected := FALSE;
         // execution finished --> set state no processing
         #statFBState := #FB_STATE_NO_PROCESSING;
       END_IF;

     ELSIF (#statStatus = #STATUS_DISCONNECTED) AND (#statBusy = true) THEN // Connection was terminated separately of send job
       #statConnected := FALSE;
       #statBusy := FALSE;
       // execution finished --> set state no processing
       #statFBState := #FB_STATE_NO_PROCESSING;

     ELSIF (#statStatus.%X15 = true) AND (#statError = false) THEN // Error occurred (#statStatus is 16#8000 to 16#FFFF)
       #statConnected := false;
       #statDone := false;
       #statBusy := false;
       #statError := true;
       #statSend.connect := false; // After error, connection is always terminated
       #statSend.req := false;
       #statTimeoutIn := false;
       // Write diagnostics
       #diagnostics.status := #statStatus;
       #diagnostics.subfunctionStatus := #statSubfunctionStatus;
       #diagnostics.stateNumber := #statFBState;
       // execution aborted --> set state no processing
       #statFBState := #FB_STATE_NO_PROCESSING;

     ELSIF ((#execute = false) AND ((#statDone = true) OR (#statError = true)))
       OR ((#statStatus = #STATUS_DISCONNECTED) AND (#statBusy = false)) // Connection was terminated separately of send job
     THEN // Reset outputs
       #statDone := false;
       #statBusy := false;
       #statError := false;
       #statResponseCode := 0;
       #statLength := 0;
       #statContentLength := 0;
       #statChunkLen := 0;
       #statEncoding := '';
       #statRcvdLen := 0;

       IF #statConnected THEN
         #statStatus := #STATUS_MONITORING;
       ELSE
         #statStatus := #STATUS_IDLE;
       END_IF;
     END_IF;

     // Write static values to outputs
     #connected := #statConnected;
     #done := #statDone;
     #busy := #statBusy;
     #error := #statError;
     #status := #statStatus;
     #responseCode := #statResponseCode;
     #length := #statLength;
     ENO := NOT #statError;
   END_REGION OUTPUTS
END_FUNCTION_BLOCK

// folder: Utilities

FUNCTION "LHTTP_ExtractStringFromArray" : Word   // FC2, SCL
{ S7_Optimized_Access := 'TRUE' }
VERSION : 0.1
   VAR_INPUT
      textBefore : String;   // Text before text that is extracted
      textAfter : String;   // Text after text that is extracted
   END_VAR
   VAR_OUTPUT
      extractedString : String;   // Extracted string
   END_VAR
   VAR_IN_OUT
      searchIn : Array[*] of Char;   // Array of Char to search in
   END_VAR
   VAR_TEMP
      tempLowerBound : DInt;   // Lower bound of given array
      tempNumElements : UDInt;   // Number of elements in given array
      tempPosInArray : DInt;   // Position in array during search
      tempLenTextBefore : Int;   // Length of text before
      tempPosTextBefore : DInt;   // Position of text before in array of Char
      tempLenTextAfter : Int;   // Length of text after
      tempPosTextAfter : Int;   // Position of text after in converted string
      tempString : String;   // Temporary string to work with
   END_VAR
   // Ret_Val : Return value; 16#0000: Successful, text was found, 16#9001: Unsuccessful, only start text was found, extracted String is filled with characters after start text, 16#9002: Unsuccessful, neither text was found
   VAR CONSTANT
      LEN_STRING : UInt := 254;   // Max. length of String
      STATUS_TEXT_FOUND : Word := 16#0000;   // Texts before and after were found
      STATUS_ONLY_START : Word := 16#9001;   // Only text before was found
      STATUS_NOTHING_FOUND : Word := 16#9002;   // Neither text was found
   END_VAR
BEGIN
   //=============================================================================
   // SIEMENS AG
   // (c)Copyright 2019
   //-----------------------------------------------------------------------------
   // Library:       LHTTP
   // Tested with:   CPU 1516-3 PN/DP V2.6
   // Engineering:   TIA Portal V15.1
   // Restrictions:  --
   // Requirements:  --
   // Functionality: Extracts a String specified by a text before and after
   //                from an array of Char
   //-----------------------------------------------------------------------------
   // Change log table:
   // Version    Date         Expert in charge         Changes applied
   // 01.00.00   01.04.2019   Siemens Online Support   First released version
   //=============================================================================

   // Initialization
   #tempPosTextBefore := 0;
   #tempPosTextAfter := 0;
   #tempLenTextBefore := LEN(#textBefore);
   #tempLenTextAfter := LEN(#textAfter);
   #extractedString := '';
   #LHTTP_ExtractStringFromArray := #STATUS_NOTHING_FOUND;

   // Get number of elements
   #tempPosInArray := #tempLowerBound := LOWER_BOUND(ARR := #searchIn, DIM := 1);
   #tempNumElements := DINT_TO_UDINT(UPPER_BOUND(ARR := #searchIn, DIM := 1) - #tempLowerBound + 1);


   // Search for text before until something was found
   REPEAT

     // Convert Chars to String
     Chars_TO_Strg(Chars  := #searchIn,
                   pChars := #tempPosInArray - #tempLowerBound, // Subtract offset since pChars is zero based
                   Cnt    := UDINT_TO_UINT(MIN(IN1 := #LEN_STRING, IN2 := #tempNumElements)),
                   Strg   => #tempString);

     // Search for text before
     #tempPosTextBefore := FIND(IN1 := #tempString, IN2 := #textBefore);

     // Text before was found
     IF #tempPosTextBefore > 0 THEN

       // Set position in array to end of text before
       #tempPosInArray += #tempPosTextBefore + #tempLenTextBefore - 1;

       // Create new string from end of text before
       Chars_TO_Strg(Chars  := #searchIn,
                     pChars := #tempPosInArray - #tempLowerBound, // Subtract offset since pChars is zero based
                     Cnt    := UDINT_TO_UINT(MIN(IN1 := #LEN_STRING, IN2 := #tempNumElements)),
                     Strg   => #tempString);

       // Find end of string to be extracted
       #tempPosTextAfter := FIND(IN1 := #tempString, IN2 := #textAfter);

       IF #tempPosTextAfter > 0 THEN // Shorten string if text after was found

         #extractedString := LEFT(IN := #tempString, L := #tempPosTextAfter - 1);
         #LHTTP_ExtractStringFromArray := #STATUS_TEXT_FOUND;
         EXIT;

       ELSE // Output whole string if text after was not found

         #extractedString := #tempString;
         #LHTTP_ExtractStringFromArray := #STATUS_ONLY_START;
         EXIT;

       END_IF;

     ELSE
       // Otherwise continue search in next string minus length of text before to ensure
       // keywords are not broken up at the end of a string and thus missed
       #tempPosInArray += UINT_TO_INT(#LEN_STRING) - #tempLenTextBefore;
     END_IF;

     // Repeat until end of array is reached
   UNTIL (#tempPosInArray > #tempNumElements) END_REPEAT;
END_FUNCTION

FUNCTION "LHTTP_FindStringInArray" : DInt   // FC5, SCL
{ S7_Optimized_Access := 'TRUE' }
VERSION : 0.1
   VAR_INPUT
      searchFor : String;   // Text that is searched for
   END_VAR
   VAR_IN_OUT
      searchIn : Array[*] of Char;   // Array of Char to search in
   END_VAR
   VAR_TEMP
      tempLowerBound : DInt;   // Lower bound of given array
      tempNumElements : UDInt;   // Number of elements in given array
      tempLenSearchFor : Int;   // Length of text that is seached for
      tempPosInArray : DInt;   // Position in array during search (0-based)
      tempPosInString : Int;   // Position in working string during search
      tempString : String;   // Temporary string to work with
   END_VAR
   // Ret_Val : Position (index) of the first character of the text that is searched for within the array of Char
   VAR CONSTANT
      LEN_STRING : UInt := 254;   // Max. length of String
   END_VAR
BEGIN
   //=============================================================================
   // SIEMENS AG
   // (c)Copyright 2019
   //-----------------------------------------------------------------------------
   // Library:       LHTTP
   // Tested with:   CPU 1516-3 PN/DP V2.6
   // Engineering:   TIA Portal V15.1
   // Restrictions:  --
   // Requirements:  --
   // Functionality: Searches for a specified String within an array of Char
   //-----------------------------------------------------------------------------
   // Change log table:
   // Version    Date         Expert in charge         Changes applied
   // 01.00.00   01.01.2019   Siemens Online Support   First released version
   //=============================================================================

   // Initialization
   #tempPosInString := 0;
   #tempPosInArray := 0;
   #tempLenSearchFor := LEN(#searchFor);
   #LHTTP_FindStringInArray := -1;

   // Get number of elements
   #tempLowerBound := LOWER_BOUND(ARR := #searchIn, DIM := 1);
   #tempNumElements := DINT_TO_UDINT(UPPER_BOUND(ARR := #searchIn, DIM := 1) - #tempLowerBound + 1);

   // Search for beginning of text until something was found
   REPEAT

     // Convert Chars to String
     Chars_TO_Strg(Chars := #searchIn,
                   pChars := #tempPosInArray,
                   Cnt := UDINT_TO_UINT(MIN(IN1 := #LEN_STRING, IN2 := #tempNumElements)),
                   Strg => #tempString);

     // Search for text at beginning
     #tempPosInString := FIND(IN1 := #tempString, IN2 := #searchFor);

     // Keyword was found
     IF #tempPosInString > 0 THEN
       // Output position of string
       #LHTTP_FindStringInArray := #tempLowerBound + #tempPosInArray + #tempPosInString - 1;
       EXIT;
     ELSE
       // Otherwise continue search in next string minus length of text at beginning to ensure
       // keywords are not broken up at the end of a string and thus missed
       #tempPosInArray += UINT_TO_INT(#LEN_STRING) - #tempLenSearchFor;
     END_IF;

   UNTIL (#tempPosInString > 0) OR (#tempPosInArray > #tempNumElements) END_REPEAT;
END_FUNCTION